FUNCTION StringToAny
VAR_INPUT
	text : T_MaxString;
	output : ANY;
END_VAR

StringToAnyType(text, output);

END_FUNCTION

(* stored: Version 1.1.0.1
   POU StringToAny: Id {c5971ef8-45ec-4504-93e7-bc3ce7d79625}, SpecialFunc None *)
